ABB RobotStudio station: Solution.rsstn

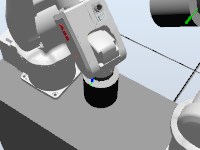
Station Solution (saved by RobotStudio 7.0.8743.626)
Controller Controller, task T_ROB3: task frame (RAPID world) sits at (-300, 0, 800) mm in the station
Controller Controller, task T_ROB2: task frame (RAPID world) sits at (-300, 0, 800) mm in the station
Controller Controller, task T_ROB1: task frame (RAPID world) sits at (-300, 0, 800) mm in the station
Controller Controller
  mechanical unit ROB_1: IRB120_3_58__01, 6 joints, base frame (0, 0, 0) mm
  mechanical unit ROB_2: IRB120_3_58__01_2, 6 joints, base frame (600, 0, 0) mm, rotated rx 0 ry 0 rz -180 deg
  mechanical unit ROB_3: IRB760_450_318__01, 6 joints, base frame (-150, 2800, -800) mm
Layout (positions relative to the parent item):
  - IRB120_3_58__01 [mechanism, from Robots\IRB120_3_58_G_01.rslib] at (-300, 0, 800) mm; joint values [-0.3299, 0.1699, 0.6158, 0, 0.7852, -0.3299] (rad or m)
  - IRB120_3_58__01_2 [mechanism, from Robots\IRB120_3_58_G_01.rslib] at (300, 0, 800) mm, rotated rx 0 ry 0 rz 180 deg; joint values [0, -0.8735, 0.5338, 0, 0.8632, 0] (rad or m)
  - IRB760_450_318__01 [mechanism, from Robots\IRB760_450_318__01.rslib] at (-450, 2800, 0) mm; joint values [0, -0.4867, -0.1103, 0] (rad or m)
  - Part_1 [part] at (-515, -200, 0) mm
  - Tool_1 [mechanism] at (-8, -100, 1120) mm, rotated rx -180 ry 0 rz 180 deg
      TCP Tool_1 at (0, 0, 0) mm
      links: SimpleGripper
  - Tool_2 [mechanism] at (183.19, 0, 1394) mm, rotated rx 180 ry 60 rz 0 deg
      TCP Tool_2 at (0, 0, 0) mm
      links: SimpleGripper
  - Tool_3 [mechanism] at (883.1, 2800, 1824.5) mm, rotated rx 180 ry 0 rz 180 deg
      TCP Tool_3 at (0, 0, 0) mm
      links: SimpleGripper
Attachment: Tool_1 is attached to IRB120_3_58__01 / Link6
Attachment: Tool_2 is attached to IRB120_3_58__01_2 / Link6
Attachment: Tool_3 is attached to IRB760_450_318__01 / Link6
Targets, tools, work objects and paths stored in the station, written as RAPID:
! task T_ROB1
MODULE CalibData
  PERS tooldata Tool_1:=[TRUE,[[0,0,0],[1,0,0,0]],[1,[0,0,1],[1,0,0,0],0,0,0]];
ENDMODULE

! task T_ROB1
MODULE Module1
  CONST robtarget AboveBeer:=[[299.255023414,-150.560096656,415.526169225],[0.0007034,-0.000000025,0.999999753,0.000000007],[-1,0,-1,0],[9E+09,9E+09,9E+09,9E+09,9E+09,9E+09]];
  CONST robtarget AtRobot1:=[[114.525825364,-5.299519863,594.446983349],[0.000703396,-0.00000003,0.999999753,0.000000009],[-1,0,-1,0],[9E+09,9E+09,9E+09,9E+09,9E+09,9E+09]];
  CONST robtarget AtBeer:=[[292,-100,320],[0,0,0,1],[-1,0,-1,0],[9E+09,9E+09,9E+09,9E+09,9E+09,9E+09]];
  PROC Path_10()
    MoveL AtRobot1,v1000,z100,Tool_1\WObj:=wobj0;
    MoveL AtBeer,v1000,z100,Tool_1\WObj:=wobj0;
  ENDPROC
ENDMODULE

! task T_ROB2
MODULE CalibData
  PERS tooldata Tool_2:=[TRUE,[[0,0,0],[1,0,0,0]],[1,[0,0,1],[1,0,0,0],0,0,0]];
ENDMODULE

! task T_ROB3
MODULE CalibData
  PERS tooldata Tool_3:=[TRUE,[[0,0,0],[1,0,0,0]],[1,[0,0,1],[1,0,0,0],0,0,0]];
ENDMODULE

